// TwinCAT 3 PLC project FMTypes
// Title: FM Types
// Company: FrameworkMonorepo
// ProjectVersion: 0.0.1
// ProgramVersion: 3.1.4024.0
// libraries:
//   Tc2_System, * (Beckhoff Automation GmbH)
//   Tc2_Utilities, * (Beckhoff Automation GmbH)
//   Tc3_JsonXml, * (Beckhoff Automation GmbH)
//   Base Interfaces,newest,System
// project tree:
//   Any/ AnyTypeUnion.TcDUT, ToAnyType.TcPOU (not stored), IsAnyTypeBound.TcPOU
//   Binding/ BoolBindingReadOnly.TcPOU, BoolBindable.TcIO, NotBind.TcPOU, Bind.TcPOU
//   Disposable/ Disposable.TcIO (not stored)
//   Numbers/ Integer.TcDUT, Decimal.TcDUT (not stored), Positive.TcDUT (not stored)
//   Queryable/ Queryable.TcIO
//   Reflection/ Reflection.TcPOU (not stored)
//   Values/BooleanExpression/ BooleanOperator.TcDUT, BooleanExpression.TcPOU
//   Values/BooleanExpression/Functions/ And2.TcPOU (not stored), And3.TcPOU, And4.TcPOU (not stored), Or2.TcPOU, Or3.TcPOU (not stored), Or4.TcPOU, Xor2.TcPOU (not stored), Xor3.TcPOU, Xor4.TcPOU
//   Values/ BoolValues.TcGVL, FalseBoolValue.TcPOU (not stored), TrueBoolValue.TcPOU, BoolValue.TcIO (not stored)
//   Version/ Global_Version.TcGVL
// real-time tasks:
//   TASK BindingTestTask: cycle T#1ms, priority 20, ADS port 350
//   TASK PlcTask: cycle T#1ms, priority 21, ADS port 351
//   TASK PlcTask1: cycle T#1ms, priority 22, ADS port 352
//   TASK PlcTask2: cycle T#1ms, priority 23, ADS port 353
//   TASK MathTestTask: cycle T#1ms, priority 24, ADS port 354
//   TASK TimesTestsTask: cycle T#1ms, priority 25, ADS port 355

// ---- Any/AnyTypeUnion.TcDUT
TYPE AnyTypeUnion :
UNION
	BOOL_ : BOOL;
	BYTE_ : BYTE;
	WORD_ : WORD;
	DWORD_ : DWORD;
	LWORD_ : LWORD;
	SINT_ : SINT;
	INT_ : INT;
	DINT_ : DINT;
	LINT_ : LINT;
	USINT_ : USINT;
	UINT_ : UINT;
	UDINT_ : UDINT;
	ULINT_ : ULINT;
	REAL_ : REAL;
	LREAL_ : LREAL;
	STRING_ : T_MaxString;
	TIME_ : TIME;
	DATE_ : DATE;
	DATEANDTIME_ : DATE_AND_TIME;
	TIMEOFDAY_ : TIME_OF_DAY;
	POINTER_ : POINTER TO BYTE;
	LTIME_ : LTIME;
END_UNION
END_TYPE

// ---- Numbers/Integer.TcDUT
TYPE Integer : LINT; END_TYPE

// ---- Values/BooleanExpression/BooleanOperator.TcDUT
{attribute 'qualified_only'}
{attribute 'strict'}
{attribute 'to_string'}
TYPE BooleanOperator :
(
	ANDop,
	ORop,
	XORop
);
END_TYPE

// ---- Values/BoolValues.TcGVL
{attribute 'qualified_only'}
VAR_GLOBAL CONSTANT
	FalseValue : FalseBoolValue := ();
	TrueValue : TrueBoolValue := ();
END_VAR

// ---- Version/Global_Version.TcGVL
{attribute 'TcGenerated'}
{attribute 'no-analysis'}
{attribute 'linkalways'}
// This function has been automatically generated from the project information.
VAR_GLOBAL CONSTANT
	{attribute 'const_non_replaced'}
	stLibVersion_FM_Types : ST_LibVersion := (iMajor := 0, iMinor := 0, iBuild := 1, iRevision := 0, nFlags := 0, sVersion := '0.0.1');
END_VAR

// ---- Binding/BoolBindable.TcIO
INTERFACE BoolBindable EXTENDS BoolValue

METHOD Bind
VAR_INPUT
	boolean : REFERENCE TO BOOL;
END_VAR
END_METHOD

{attribute 'monitoring' := 'call'}
PROPERTY IsBound : BOOL
GET
END_GET
END_PROPERTY

{attribute 'monitoring' := 'call'}
PROPERTY Value : BOOL
GET
END_GET
END_PROPERTY

END_INTERFACE

// ---- Queryable/Queryable.TcIO
INTERFACE Queryable EXTENDS __SYSTEM.IQueryInterface

END_INTERFACE

// ---- Values/TrueBoolValue.TcPOU
FUNCTION_BLOCK TrueBoolValue IMPLEMENTS BoolValue
VAR
END_VAR

{attribute 'monitoring' := 'call'}
PROPERTY Value : BOOL
GET
Value := TRUE;
END_GET
END_PROPERTY

END_FUNCTION_BLOCK

// ---- Any/IsAnyTypeBound.TcPOU
FUNCTION IsAnyTypeBound : BOOL
VAR_INPUT
	anytype : __SYSTEM.AnyType;
END_VAR

IsAnyTypeBound := anytype.pValue <> 0 AND anytype.diSize > 0;

END_FUNCTION

// ---- Binding/BoolBindingReadOnly.TcPOU
{attribute 'hide_all_locals'}
{attribute 'enable_dynamic_creation'}
FUNCTION_BLOCK BoolBindingReadOnly IMPLEMENTS BoolBindable, Disposable
VAR
	ref : REFERENCE TO BOOL;
	_Negate : BOOL;
END_VAR

METHOD Bind
VAR_INPUT
	boolean : REFERENCE TO BOOL;
END_VAR
ref REF= boolean;
END_METHOD

METHOD Dispose
__DELETE(THIS);
END_METHOD

{attribute 'monitoring' := 'call'}
PROPERTY IsBound : BOOL
GET
IsBound := __ISVALIDREF(ref);
END_GET
END_PROPERTY

PROPERTY Negate : BOOL
GET
Negate := _Negate;
END_GET
SET
_Negate := Negate;
END_SET
END_PROPERTY

{attribute 'monitoring' := 'call'}
PROPERTY Value : BOOL
GET
Value := ref XOR _Negate;
END_GET
END_PROPERTY

END_FUNCTION_BLOCK

// ---- Binding/Bind.TcPOU
FUNCTION Bind : BoolValue
VAR_INPUT
	boolean : REFERENCE TO BOOL;
END_VAR
VAR
	p : POINTER TO BoolBindingReadOnly;
END_VAR

p := __NEW(BoolBindingReadOnly);

p^.Bind(boolean);

Bind := p^;

END_FUNCTION

// ---- Binding/NotBind.TcPOU
FUNCTION NotBind : BoolValue
VAR_INPUT
	boolean : REFERENCE TO BOOL;
END_VAR
VAR
	p : POINTER TO BoolBindingReadOnly;
END_VAR

p := __NEW(BoolBindingReadOnly);

p^.Bind(boolean);
p^.Negate := TRUE;

NotBind := p^;

END_FUNCTION

// ---- Values/BooleanExpression/BooleanExpression.TcPOU
{attribute 'hide_all_locals'}
{attribute 'enable_dynamic_creation'}
FUNCTION_BLOCK BooleanExpression IMPLEMENTS BoolValue, Disposable
VAR
	operands : ARRAY[0..MaxIndex - 1] OF BoolValue;
	operandCount : INT;
	operator : BooleanOperator;
END_VAR
VAR CONSTANT
	MaxIndex : INT := 4;
END_VAR

METHOD Clear
VAR
	i : INT;
	disposable : Disposable;
END_VAR
FOR i := 0 TO operandCount - 1 DO
	__QUERYINTERFACE(operands[i], disposable);
	disposable.Dispose();
	operands[i] := 0;
END_FOR

operandCount := 0;
END_METHOD

METHOD Dispose
VAR
	i : INT;
	disposable : Disposable;
END_VAR
Clear();
__DELETE(THIS);
END_METHOD

METHOD FB_exit : BOOL
VAR_INPUT
	bInCopyCode : BOOL; // if TRUE, the exit method is called for exiting an instance that is copied afterwards (online change).
END_VAR
Clear();
END_METHOD

METHOD Op2
VAR_INPUT
	operator : BooleanOperator;
	value1 : BoolValue;
	value2 : BoolValue;
END_VAR
Clear();

THIS^.operator := operator;

operands[0] := value1;
operands[1] := value2;
operandCount := 2;
END_METHOD

METHOD Op3
VAR_INPUT
	operator : BooleanOperator;
	value1 : BoolValue;
	value2 : BoolValue;
	value3 : BoolValue;
END_VAR
Clear();

THIS^.operator := operator;

operands[0] := value1;
operands[1] := value2;
operands[2] := value3;
operandCount := 3;
END_METHOD

METHOD Op4
VAR_INPUT
	operator : BooleanOperator;
	value1 : BoolValue;
	value2 : BoolValue;
	value3 : BoolValue;
	value4 : BoolValue;
END_VAR
Clear();

THIS^.operator := operator;

operands[0] := value1;
operands[1] := value2;
operands[2] := value3;
operands[3] := value4;
operandCount := 4;
END_METHOD

{attribute 'monitoring' := 'call'}
PROPERTY Value : BOOL
GET
VAR
	i : INT;
	result : BOOL;
END_VAR
IF (operandCount = 0) THEN
	RETURN;
END_IF

CASE operator OF
	
	BooleanOperator.ANDop:
		
		result := operands[0].Value;
		FOR i := 1 TO operandCount - 1 DO
			result := result AND operands[i].Value;
		END_FOR	
		
	BooleanOperator.ORop:
		
		result := operands[0].Value;
		FOR i := 1 TO operandCount - 1 DO
			result := result OR operands[i].Value;
		END_FOR	
		
	BooleanOperator.XORop:
		
		result := operands[0].Value;
		FOR i := 1 TO operandCount - 1 DO
			result := result XOR operands[i].Value;
		END_FOR	
		
END_CASE

Value := result;
END_GET
END_PROPERTY

END_FUNCTION_BLOCK

// ---- Values/BooleanExpression/Functions/And3.TcPOU
FUNCTION And3 : BoolValue
VAR_INPUT
	value1 : BoolValue;
	value2 : BoolValue;
	value3 : BoolValue;
END_VAR
VAR
	p : POINTER TO BooleanExpression;
END_VAR

p := __NEW(BooleanExpression);

p^.Op3(
	operator := BooleanOperator.ANDop,
	value1 := value1,
	value2 := value2,
	value3 := value3
);

And3 := p^;

END_FUNCTION

// ---- Values/BooleanExpression/Functions/Or2.TcPOU
FUNCTION Or2 : BoolValue
VAR_INPUT
	value1 : BoolValue;
	value2 : BoolValue;
END_VAR
VAR
	p : POINTER TO BooleanExpression;
END_VAR

p := __NEW(BooleanExpression);

p^.Op2(
	operator := BooleanOperator.ORop,
	value1 := value1,
	value2 := value2
);

Or2 := p^;

END_FUNCTION

// ---- Values/BooleanExpression/Functions/Or4.TcPOU
FUNCTION Or4 : BoolValue
VAR_INPUT
	value1 : BoolValue;
	value2 : BoolValue;
	value3 : BoolValue;
	value4 : BoolValue;
END_VAR
VAR
	p : POINTER TO BooleanExpression;
END_VAR

p := __NEW(BooleanExpression);

p^.Op4(
	operator := BooleanOperator.ORop,
	value1 := value1,
	value2 := value2,
	value3 := value3,
	value4 := value4
);

Or4 := p^;

END_FUNCTION

// ---- Values/BooleanExpression/Functions/Xor3.TcPOU
FUNCTION Xor3 : BoolValue
VAR_INPUT
	value1 : BoolValue;
	value2 : BoolValue;
	value3 : BoolValue;
END_VAR
VAR
	p : POINTER TO BooleanExpression;
END_VAR

p := __NEW(BooleanExpression);

p^.Op3(
	operator := BooleanOperator.XORop,
	value1 := value1,
	value2 := value2,
	value3 := value3
);

Xor3 := p^;

END_FUNCTION

// ---- Values/BooleanExpression/Functions/Xor4.TcPOU
FUNCTION Xor4 : BoolValue
VAR_INPUT
	value1 : BoolValue;
	value2 : BoolValue;
	value3 : BoolValue;
	value4 : BoolValue;
END_VAR
VAR
	p : POINTER TO BooleanExpression;
END_VAR

p := __NEW(BooleanExpression);

p^.Op4(
	operator := BooleanOperator.XORop,
	value1 := value1,
	value2 := value2,
	value3 := value3,
	value4 := value4
);

Xor4 := p^;

END_FUNCTION
